FUNCTION_BLOCK CoeReaderEx EXTENDS FB_EcCoESdoReadEx
VAR_OUTPUT
    eAdsError : TcError.AdsErrorCodes;
END_VAR

SUPER^();
eAdsError := TcError.ToAdsErrorCode(SUPER^.nErrId);

END_FUNCTION_BLOCK

(* stored: Version 1.1.0.1
   POU CoeReaderEx: Id {cb11d66a-6172-04ac-0ce8-e9577bac676c}, SpecialFunc None *)
